TYPE (* Publish event type to be sent to the EventHandler *)
  (* Standard: 61499-2; Description: Copyright (c) 2019 fortiss GmbH This program and the accompanying materials are made available under the terms of the Eclipse Public License 2.0 which is available at https://www.eclipse.org/legal/epl-2.0/ SPDX-License-Identifier: EPL-2.0 *)
  (* Version 1.0, 2019-09-17, Jose Cabral, fortiss GmbH *)
  (* ASN.1 tag APPLICATION 1 *)
  PublishEvent : STRUCT
    source : ArrowheadSystem; (* ArrowheadSystem publishing the event. *)
    event : ArrowheadEvent; (* The published event. *)
    deliveryCompleteUri : WSTRING; (* The URL subpath the Event Handler can use to inform the publisher about the results of the event propagation. If null, the Event Handler will not try to send the results. *)
  END_STRUCT;
END_TYPE
